Staubli VAL3: numericalTwins.dtx

bool bFinish
bool bOvrPosition
bool bResult = true
frame fPlateau = {x=632.308207, y=706.981098, z=-559.699722, rx=-0.00630742, ry=-0.102848, rz=-0.154308, fatherId=world[0]}
jointRx home = {j1=64, j2=-30, j3=143, j4=-103, j5=60, j6=116}
jointRx jHere = {j1=45.383273, j2=1.666947, j3=107.278201, j4=-97.512292, j5=76.926774, j6=121.888458}
jointRx jStart
mdesc mNomSpeed = {vel=50}
mdesc vitextrusion = {rmax=500, tmax=17, leave=15, reach=15}
num nAckIndex
num nCmdIndex = 4
num nCmdType = 1
num nCmdVel = 50
num nData = 10
num nDivider = 59
num nEof = 125
num nEol = 10
num nFrameIndex = 3553
num nIndexQueue[5]
  [0] = 1
  [1] = 2
  [2] = 3
  [3] = 4
num nLastIndex
num nNbChar
num nOvrPos
num nPrevOvrPos
num nQueueCount
num nQueueRead
num nQueueSize = 5
num nQueueWrite
num nSof = 123
num nTypeQueue[5]
  [0] = 1
  [1] = 1
  [2] = 1
  [3] = 1
num nVelQueue[5]
  [0] = 50
  [1] = 50
  [2] = 50
  [3] = 50
pointRx pAccostage = {x=200, y=-150, z=5, rx=-180, ry=7.016478e-15, rz=-180, fatherId=fPlateau[0]}
pointRx pChauffe = {x=-200, z=200, ry=180, fatherId=fPlateau[0]}
pointRx pCmdQueue[5]
  [0] = {x=371.256502, y=762.70159, z=186.0845966, rx=89.692992, ry=69.84956, rz=-90.0731633, shoulder=lefty, elbow=epositive, wrist=wpositive, fatherId=world[0]}
  [1] = {x=371.256502, y=762.70159, z=186.0845966, rx=89.692992, ry=69.84956, rz=-90.0731633, shoulder=lefty, elbow=epositive, wrist=wpositive, fatherId=world[0]}
  [2] = {x=371.256502, y=762.70159, z=186.0845966, rx=89.692992, ry=69.84956, rz=-90.0731633, shoulder=lefty, elbow=epositive, wrist=wpositive, fatherId=world[0]}
  [3] = {x=371.256502, y=762.70159, z=186.0845966, rx=89.692992, ry=69.84956, rz=-90.0731633, shoulder=lefty, elbow=epositive, wrist=wpositive, fatherId=world[0]}
  [4] = {x=371.256502, y=762.70159, z=186.0845966, rx=89.692992, ry=69.84956, rz=-90.0731633, shoulder=lefty, elbow=epositive, wrist=wpositive, fatherId=world[0]}
pointRx pDegagement = {z=200, ry=180, fatherId=fPlateau[0]}
pointRx pHere = {x=832.0401931, y=692.000932864, z=529.509333, rx=84.591408, ry=60.0803316, rz=-73.577687, shoulder=lefty, elbow=epositive, wrist=wpositive, fatherId=world[0]}
sio sioSocket = {link=Socket\toto}
string sAck
string sData = "{3553;    45.383;     1.667;   107.278;   -97.512;    76.927;   121.888;832.04 ;692.001;529.509;84.591;60.08 ;-73.578}"
string sDataIn
string sTaskCmd = "tCommande"
string sTaskPos = "tPosition"
string sTaskRobot = "tRobot"
tool tBuse = {x=551, y=-30, z=75, ry=90, rz=-20, fatherId=flange[0], ioLink=valve1}
tool tPalpage = {x=655.7, y=-30, z=75, ry=90, rz=-20, fatherId=flange[0]}
